PROGRAM P2_03_Production_Ctrl
VAR
	bFeeding_Active					:BOOL;
	bMixing_Active					:BOOL;
	bGranulation_Active				:BOOL;
	bDischarge_Active				:BOOL;
END_VAR

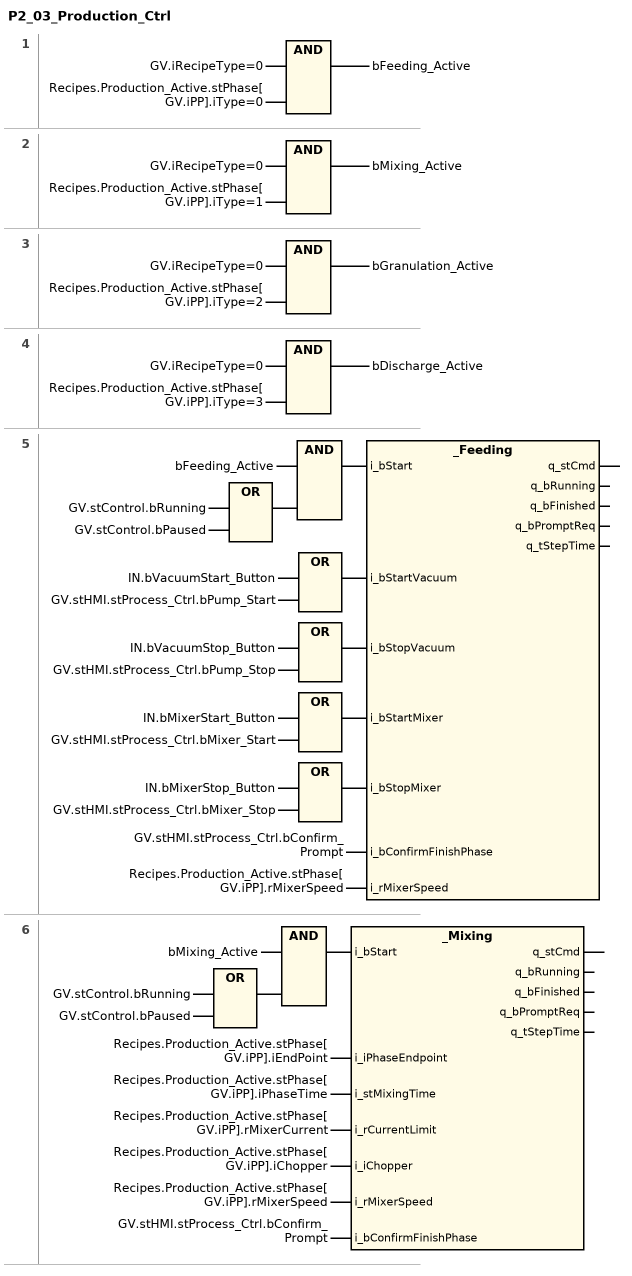
// NETWORK 1
bFeeding_Active := (GV.iRecipeType=0) AND (Recipes.Production_Active.stPhase[GV.iPP].iType=0);

// NETWORK 2
bMixing_Active := (GV.iRecipeType=0) AND (Recipes.Production_Active.stPhase[GV.iPP].iType=1);

// NETWORK 3
bGranulation_Active := (GV.iRecipeType=0) AND (Recipes.Production_Active.stPhase[GV.iPP].iType=2);

// NETWORK 4
bDischarge_Active := (GV.iRecipeType=0) AND (Recipes.Production_Active.stPhase[GV.iPP].iType=3);

// NETWORK 5
_Feeding(i_bStart := bFeeding_Active AND (GV.stControl.bRunning OR GV.stControl.bPaused), i_bStartVacuum := IN.bVacuumStart_Button OR GV.stHMI.stProcess_Ctrl.bPump_Start, i_bStopVacuum := IN.bVacuumStop_Button OR GV.stHMI.stProcess_Ctrl.bPump_Stop, i_bStartMixer := IN.bMixerStart_Button OR GV.stHMI.stProcess_Ctrl.bMixer_Start, i_bStopMixer := IN.bMixerStop_Button OR GV.stHMI.stProcess_Ctrl.bMixer_Stop, i_bConfirmFinishPhase := GV.stHMI.stProcess_Ctrl.bConfirm_Prompt, i_rMixerSpeed := Recipes.Production_Active.stPhase[GV.iPP].rMixerSpeed);

// NETWORK 6
_Mixing(i_bStart := bMixing_Active AND (GV.stControl.bRunning OR GV.stControl.bPaused), i_iPhaseEndpoint := Recipes.Production_Active.stPhase[GV.iPP].iEndPoint, i_stMixingTime := Recipes.Production_Active.stPhase[GV.iPP].iPhaseTime, i_rCurrentLimit := Recipes.Production_Active.stPhase[GV.iPP].rMixerCurrent, i_iChopper := Recipes.Production_Active.stPhase[GV.iPP].iChopper, i_rMixerSpeed := Recipes.Production_Active.stPhase[GV.iPP].rMixerSpeed, i_bConfirmFinishPhase := GV.stHMI.stProcess_Ctrl.bConfirm_Prompt);

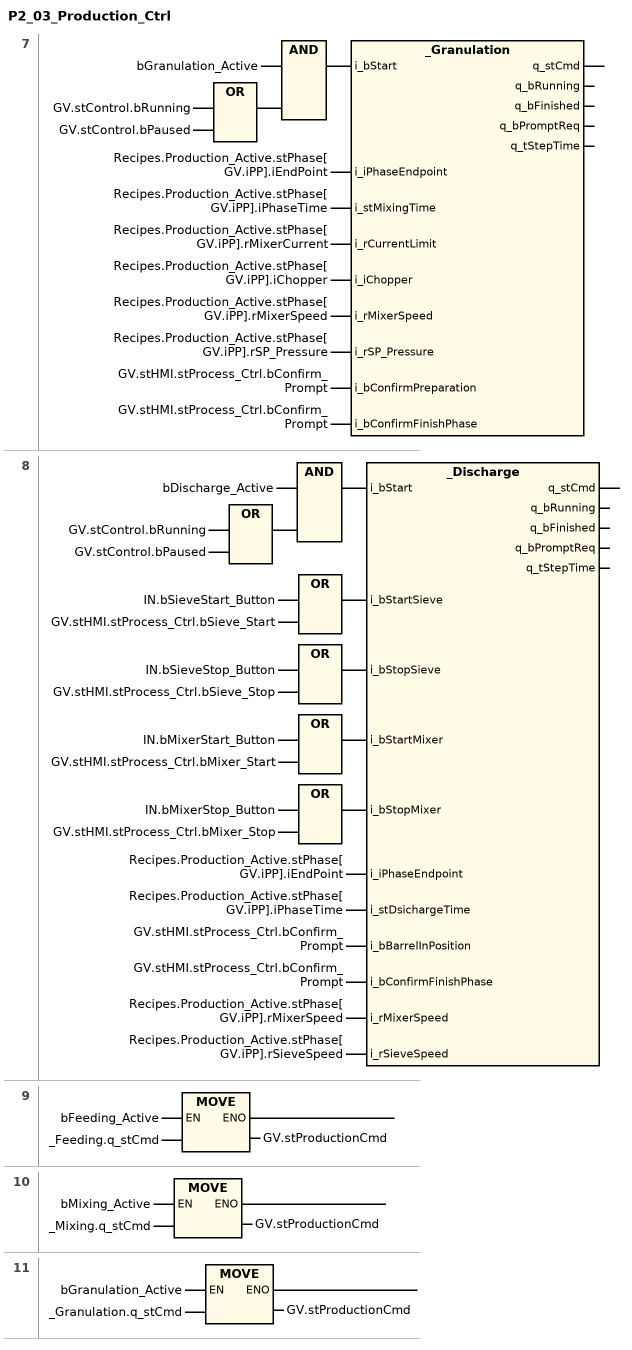
// NETWORK 7
_Granulation(i_bStart := bGranulation_Active AND (GV.stControl.bRunning OR GV.stControl.bPaused), i_iPhaseEndpoint := Recipes.Production_Active.stPhase[GV.iPP].iEndPoint, i_stMixingTime := Recipes.Production_Active.stPhase[GV.iPP].iPhaseTime, i_rCurrentLimit := Recipes.Production_Active.stPhase[GV.iPP].rMixerCurrent, i_iChopper := Recipes.Production_Active.stPhase[GV.iPP].iChopper, i_rMixerSpeed := Recipes.Production_Active.stPhase[GV.iPP].rMixerSpeed, i_rSP_Pressure := Recipes.Production_Active.stPhase[GV.iPP].rSP_Pressure, i_bConfirmPreparation := GV.stHMI.stProcess_Ctrl.bConfirm_Prompt, i_bConfirmFinishPhase := GV.stHMI.stProcess_Ctrl.bConfirm_Prompt);

// NETWORK 8
_Discharge(i_bStart := bDischarge_Active AND (GV.stControl.bRunning OR GV.stControl.bPaused), i_bStartSieve := IN.bSieveStart_Button OR GV.stHMI.stProcess_Ctrl.bSieve_Start, i_bStopSieve := IN.bSieveStop_Button OR GV.stHMI.stProcess_Ctrl.bSieve_Stop, i_bStartMixer := IN.bMixerStart_Button OR GV.stHMI.stProcess_Ctrl.bMixer_Start, i_bStopMixer := IN.bMixerStop_Button OR GV.stHMI.stProcess_Ctrl.bMixer_Stop, i_iPhaseEndpoint := Recipes.Production_Active.stPhase[GV.iPP].iEndPoint, i_stDsichargeTime := Recipes.Production_Active.stPhase[GV.iPP].iPhaseTime, i_bBarrelInPosition := GV.stHMI.stProcess_Ctrl.bConfirm_Prompt, i_bConfirmFinishPhase := GV.stHMI.stProcess_Ctrl.bConfirm_Prompt, i_rMixerSpeed := Recipes.Production_Active.stPhase[GV.iPP].rMixerSpeed, i_rSieveSpeed := Recipes.Production_Active.stPhase[GV.iPP].rSieveSpeed);

// NETWORK 9
IF bFeeding_Active THEN GV.stProductionCmd := _Feeding.q_stCmd; END_IF

// NETWORK 10
IF bMixing_Active THEN GV.stProductionCmd := _Mixing.q_stCmd; END_IF

// NETWORK 11
IF bGranulation_Active THEN GV.stProductionCmd := _Granulation.q_stCmd; END_IF

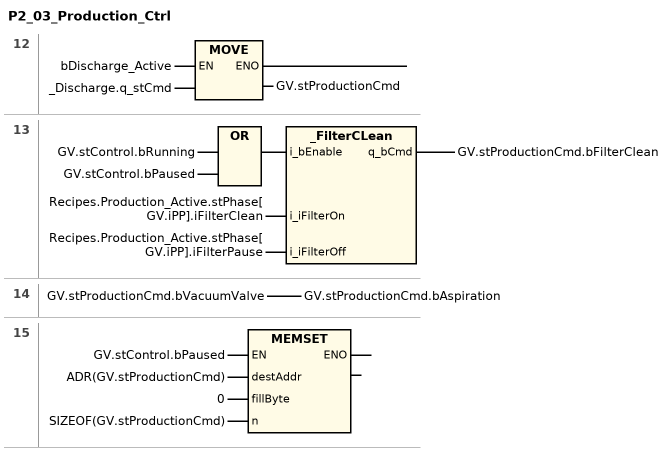
// NETWORK 12
IF bDischarge_Active THEN GV.stProductionCmd := _Discharge.q_stCmd; END_IF

// NETWORK 13
_FilterCLean(i_bEnable := GV.stControl.bRunning OR GV.stControl.bPaused, i_iFilterOn := Recipes.Production_Active.stPhase[GV.iPP].iFilterClean, i_iFilterOff := Recipes.Production_Active.stPhase[GV.iPP].iFilterPause);
GV.stProductionCmd.bFilterClean := _FilterCLean.q_bCmd;

// NETWORK 14
GV.stProductionCmd.bAspiration := GV.stProductionCmd.bVacuumValve;

// NETWORK 15
IF GV.stControl.bPaused THEN
    MEMSET(destAddr := ADR(GV.stProductionCmd), fillByte := 0, n := SIZEOF(GV.stProductionCmd));
END_IF

END_PROGRAM

(* stored: Version 1.1.0.1, ProductVersion 3.1.4026.13
   POU P2_03_Production_Ctrl: Id {e40e2bd6-ef31-4d1b-b941-ee222a4b302b}, SpecialFunc None *)
